FUNCTION_BLOCK TcCommand IMPLEMENTS itfCommand
//VAR_INPUT
//END_VAR
//VAR_OUTPUT
//END_VAR
VAR
	_Command        : ST_Command;	
END_VAR

{warning 'add method implementation '}
METHOD Abort : MC_Error
VAR
	
END_VAR
END_METHOD

{warning 'add property implementation'}
PROPERTY Active : BOOL
GET
Active := _Command.Active;
END_GET
SET
_Command.Active := Active;
END_SET
END_PROPERTY

{warning 'add property implementation'}
PROPERTY Busy : BOOL
GET
Busy := _Command.Busy;
END_GET
SET
_Command.Busy := Busy;
END_SET
END_PROPERTY

{warning 'add property implementation'}
PROPERTY Command : MC_COMMAND_REF
GET
Command := _Command.Command;
END_GET
SET
 _Command.Command :=  Command;
END_SET
END_PROPERTY

{warning 'add property implementation'}
PROPERTY CommandAborted : BOOL
GET
CommandAborted := _Command.CommandAborted;
END_GET
SET
 _Command.CommandAborted := CommandAborted;
END_SET
END_PROPERTY

{warning 'add property implementation'}
PROPERTY Done : BOOL
GET
Done := _Command.Done;
END_GET
SET
_Command.Done := Done;
END_SET
END_PROPERTY

{warning 'add property implementation'}
PROPERTY Error : BOOL
GET
Error := _Command.Error;
END_GET
SET
_Command.Error := Error;
END_SET
END_PROPERTY

{warning 'add property implementation'}
PROPERTY ErrorId : MC_Error
GET
ErrorId := _Command.ErrorId;
END_GET
SET
_Command.ErrorId := ErrorId;
END_SET
END_PROPERTY

PROPERTY ErrorID_Udint : UDINT
GET
ErrorID_Udint := _Command.ErrorID_Udint;
END_GET
SET
_Command.ErrorID_Udint := ErrorID_Udint;
END_SET
END_PROPERTY

{warning 'add method implementation '}
METHOD Wait : MC_Error (* This method only makes sense in the IEC 61499 environment*)
VAR_INPUT
	Timeout	: TIME;
	AbortOnTimeout	: BOOL;
END_VAR
VAR
	
END_VAR
END_METHOD

END_FUNCTION_BLOCK

(* stored: Version 1.1.0.1, ProductVersion 3.1.4024.12
   POU TcCommand: Id {e8f9fb2a-654e-4cba-815b-553b67545df0}, SpecialFunc None
   Method Abort: Id {24a343c7-760a-41b7-bb70-f72b5e25b299}
   Property Active: Id {2720e767-fe04-44c0-bbcf-f06184d2ad20}
   Get Get: Id {b11ca942-0adc-4d97-80c8-4668e727e494}
   Set Set: Id {32c544ad-fa82-4c92-80c2-55828e34d554}
   Property Busy: Id {cf8f3abf-9327-4e38-ac9d-65ef09dc1f16}
   Get Get: Id {2c33ef5d-6052-4199-ac6a-ec7a8a9b5029}
   Set Set: Id {3e8d634e-f252-4264-8411-8fe4ce317e8b}
   Property Command: Id {378c910e-a8c7-4401-9098-8e04a5ab9cd3}
   Get Get: Id {80d78255-7df6-47d0-99a3-fd5ea2122407}
   Set Set: Id {e9b0ea02-628f-4ba0-90c1-5a1ff9d57d74}
   Property CommandAborted: Id {e97f9496-7981-4895-aa93-8dab67642603}
   Get Get: Id {6cdf14cb-71eb-4a12-8464-a204bbfa90a9}
   Set Set: Id {b5f29b6d-2575-413d-b9a0-e54c27480445}
   Property Done: Id {357dca3d-7954-47ca-bf93-29e0741b485f}
   Get Get: Id {270c9587-1b81-49c6-8750-d802bc67f571}
   Set Set: Id {ed4328b7-b43d-4f76-ade7-db01b701244c}
   Property Error: Id {8340cbd2-7fc3-4229-8fbe-a3ec0ac74ef3}
   Get Get: Id {801043b3-ef60-452f-ab45-3caaf23495cb}
   Set Set: Id {97167a2d-0425-42b3-ac16-7f070b5b016a}
   Property ErrorId: Id {fe72e8ec-5584-486b-a73a-dafdbeb5627c}
   Get Get: Id {174e5abd-8e7a-4372-ac8c-f261dc1ba5b8}
   Set Set: Id {72fcc745-c329-48e5-af68-49e95ba9f03e}
   Property ErrorID_Udint: Id {554ee8f6-4246-4f19-9a2a-a20d45173f83}
   Get Get: Id {7db93102-df1d-40a5-b5b8-3dbce321da57}
   Set Set: Id {e7001d4d-398b-43ec-9350-fc1bdca27ab7}
   Method Wait: Id {9f601dc2-318f-45fa-99c9-69984c49fb48} *)
